{attribute 'qualified_only'}
{attribute 'strict'}
TYPE ENUM_EpicsHomeCmd :
(
	EPICS_MOTOR_HOME_LLS := 1, // Low limit switch
	EPICS_MOTOR_HOME_HLS := 2, // High limit switch
	EPICS_MOTOR_HOME_LHS := 3, // Home switch via low switch
	EPICS_MOTOR_HOME_HHS := 4, // Home switch via high switch
	EPICS_MOTOR_HOME_ABS := 15, // Set here to be fHomePosition
	EPICS_MOTOR_HOME_NONE := -1 // Do not home, ever
);
END_TYPE

(* stored: Version 1.1.0.1, ProductVersion 3.1.4020.14
   DUT ENUM_EpicsHomeCmd: Id {97391387-6673-4061-a135-1a0002888344} *)
